// TwinCAT 3 PLC project CraneSimulation
// ProgramVersion: 3.1.4023.0
// libraries:
//   Tc2_Standard, * (Beckhoff Automation GmbH)
//   Tc2_System, * (Beckhoff Automation GmbH)
//   Tc3_Module, * (Beckhoff Automation GmbH)
//   VisuDialogs, * (System)
//   VisuSymbols,3.5.10.0,System
// project tree:
//   DUTs/ E_CraneMode.TcDUT, E_CraneStatus.TcDUT, E_ErrorModes.TcDUT, ST_CraneKinematics.TcDUT (not stored), ST_CraneParameters.TcDUT, ST_PistonOutOfBounds.TcDUT, ST_PistonRange.TcDUT, ST_StateVariables.TcDUT
//   / GlobalTextList.TcGTLO, PlcTask.TcTTO (not stored), Visualization Manager.TcVMO (not stored)
//   GVLs/ HMI.TcGVL, Inputs.TcGVL, Outputs.TcGVL, Parameters.TcGVL
//   POUs/ CraneSimulation.TcPOU, MAIN.TcPOU
//   POUs/Function blocks/ FB_AutomaticControl.TcPOU, FB_CheckPistonPosition.TcPOU, FB_CraneMode.TcPOU, FB_CraneStatus.TcPOU, FB_ManualControl.TcPOU, FB_MotionReferenceGenerator.TcPOU, FB_OpenLoopControl.TcPOU
//   POUs/Functions/ F_BarToPascal.TcPOU, F_BoomAngle.TcPOU, F_CheckPistonPosition.TcPOU, F_LminToSI.TcPOU, F_PistonDisplacementToBoomAngle.TcPOU, F_RadToDeg.TcPOU
//   VISUs/ CraneSimulationHMI.TcVIS

// ---- DUTs/E_CraneMode.TcDUT
{attribute 'qualified_only'}
{attribute 'strict'}
TYPE E_CraneMode :
(
	Manual,
	Automatic,
	NaN
);
END_TYPE

// ---- DUTs/E_CraneStatus.TcDUT
{attribute 'qualified_only'}
{attribute 'strict'}
TYPE E_CraneStatus :
(
	Error,
	Ready,
	Running,
	Stopping,
	PowerOff,
	Checking
);
END_TYPE

// ---- DUTs/E_ErrorModes.TcDUT
{attribute 'qualified_only'}
{attribute 'strict'}
TYPE E_ErrorModes :
(
	NaN,
	MaxLimit,
	MinLimit
);
END_TYPE

// ---- DUTs/ST_CraneParameters.TcDUT
TYPE ST_CraneParameters :
STRUCT
	fCyclicTime : LREAL := 0.01; //[s]
	fMaxVelocityLimit : LREAL := 0.05; //[m/s]
	fBoreArea : LREAL := 0.0033183;
	fAnnulusArea : LREAL := 0.0023562;
	fMaxFlowCapacity : LREAL := 30; //[l/min]
END_STRUCT
END_TYPE

// ---- DUTs/ST_PistonOutOfBounds.TcDUT
TYPE ST_PistonOutOfBounds :
STRUCT
	sNotActive : STRING := 'End Stop not active';
	sPistonMax : STRING := 'Piston has reached upper end stop';
	sPistonMin : STRING := 'Piston has reached lower end stop';
END_STRUCT
END_TYPE

// ---- DUTs/ST_PistonRange.TcDUT
TYPE ST_PistonRange :
STRUCT
	fPistonPosMax : REAL := 0.5;
	fPistonPosMin : REAL := 0.0;
END_STRUCT
END_TYPE

// ---- DUTs/ST_StateVariables.TcDUT
TYPE ST_StateVariables :
STRUCT
	bPower : BOOL;
	bStart : BOOL;
	bStop : BOOL;
	bRunning : BOOL := FALSE;
	bError : BOOL;
	bMode : BOOL;
	fTime : LREAL := 0.0;
END_STRUCT
END_TYPE

// ---- GVLs/HMI.TcGVL
{attribute 'qualified_only'}
VAR_GLOBAL
	fManualCylinderPositionReference : LREAL;
	sPistonEndStopMessage : STRING;
	fCylinderPositonReference : LREAL := 0.0;
	fCylinderVelocityReference : LREAL := 0.0;
	fBoomAngle : LREAL;
END_VAR

// ---- GVLs/Inputs.TcGVL
{attribute 'qualified_only'}
VAR_GLOBAL
	bOnSelector : BOOL;
	bAutoSelector : BOOL;
	bStartButton : BOOL;
	bStopButton : BOOL;
	fJoystickX : LREAL;
	fJoystickY : LREAL;
END_VAR

// ---- GVLs/Outputs.TcGVL
{attribute 'qualified_only'}
VAR_GLOBAL
	bStartLight : BOOL;
	bStopLight : BOOL;
	eCraneMode : E_CraneMode;
	eCraneStatus : E_CraneStatus;
	fOutputVelocity : LREAL;
END_VAR

// ---- GVLs/Parameters.TcGVL
{attribute 'qualified_only'}
VAR_GLOBAL
	fCyclicTime : REAL := 0.01;
	bSimulationRunning : BOOL := FALSE;
	stPistonRange : ST_PistonRange;
	stPistonOutOfBounds : ST_PistonOutOfBounds;
	stCraneKinematics : ST_CraneKinematics;
	stStateVariables : ST_StateVariables;
	stCraneParameters : ST_CraneParameters;
	eErrorModes : E_ErrorModes;
END_VAR

// ---- POUs/CraneSimulation.TcPOU
PROGRAM CraneSimulation
VAR
	fCyclicTime : LREAL := 0.01;
	
	fbCraneStatus : FB_CraneStatus;
	fbCraneMode : FB_CraneMode;
END_VAR

// Crane status state machine
fbCraneStatus(	bPower := Inputs.bOnSelector,
		 		bStart := Inputs.bStartButton, 
				bStop := Inputs.bStopButton, 
				bRunning := Parameters.stStateVariables.bRunning, 
				bError := Parameters.stStateVariables.bError,
				eCraneStatus => Outputs.eCraneStatus);

// Crane mode state machine
IF Parameters.stStateVariables.bRunning THEN
	fbCraneMode( 	bRunning := Parameters.stStateVariables.bRunning,
					bMode := Inputs.bAutoSelector,
					eCraneMode => Outputs.eCraneMode);
END_IF
	
// Calculate boom angle for visualization of simulation		
HMI.fBoomAngle := F_BoomAngle(	fCylinderX := HMI.fCylinderPositonReference);

// Simulation timer			
IF Parameters.stStateVariables.bRunning THEN
	Parameters.stStateVariables.fTime := Parameters.stStateVariables.fTime + fCyclicTime;
ELSE
	Parameters.stStateVariables.fTime := 0.0;
END_IF

END_PROGRAM

// ---- POUs/Function blocks/FB_CraneStatus.TcPOU
FUNCTION_BLOCK FB_CraneStatus
VAR_INPUT
	bPower : BOOL;
	bStart : BOOL;
	bStop : BOOL;
	bRunning : BOOL;
	bError : BOOL;
END_VAR
VAR_OUTPUT
	eCraneStatus : E_CraneStatus := E_CraneStatus.PowerOff;
END_VAR
VAR
END_VAR

//Status state machine
CASE eCraneStatus OF
	E_CraneStatus.PowerOff:
		IF bPower THEN
			eCraneStatus := E_CraneStatus.Checking;
		END_IF	
	
	E_CraneStatus.Error:
		Outputs.bStopLight := TRUE;
		
		IF NOT bError THEN
			eCraneStatus := E_CraneStatus.Checking;
		END_IF
		
	E_CraneStatus.Checking:
		Outputs.bStopLight := FALSE;
		Outputs.bStartLight := FALSE;
		
		IF (NOT bError) THEN
			eCraneStatus := E_CraneStatus.Ready;
		ELSE
			eCraneStatus := E_CraneStatus.Error;
		END_IF
		
		IF bPower AND NOT bError THEN
			eCraneStatus := E_CraneStatus.Ready;
		ELSE
			eCraneStatus := E_CraneStatus.PowerOff;
		END_IF
		
	E_CraneStatus.Ready:
		IF bStart AND bPower AND NOT(bError) THEN
			Parameters.stStateVariables.bRunning := TRUE;
			Parameters.stStateVariables.bStart := FALSE;
			eCraneStatus := E_CraneStatus.Running;
		END_IF	
		
		IF  NOT(bPower) OR bError THEN
			eCraneStatus := E_CraneStatus.Checking;
		END_IF	
		
	E_CraneStatus.Running:
		Outputs.bStartLight := TRUE;
		
		F_CheckPistonPosition();
		
		IF bStop THEN
			eCraneStatus := E_CraneStatus.Stopping;
		END_IF
		
		IF bError OR NOT bRunning OR NOT bPOWER THEN
			eCraneStatus := E_CraneStatus.Checking;
		END_IF
		
	E_CraneStatus.Stopping:
		Parameters.stStateVariables.bRunning := FALSE;
		Parameters.stStateVariables.bStart := FALSE;
		Outputs.bStopLight := TRUE;
	
		IF NOT bRunning OR bPower OR bError THEN
			eCraneStatus := E_CraneStatus.Checking;
		END_IF
	ELSE
		eCraneStatus := E_CraneStatus.Checking;
		
END_CASE

END_FUNCTION_BLOCK

// ---- POUs/Functions/F_CheckPistonPosition.TcPOU
FUNCTION F_CheckPistonPosition : E_ErrorModes
VAR_INPUT
END_VAR
VAR
END_VAR

// Check if piston is out of bounds
IF HMI.fCylinderPositonReference > Parameters.stPistonRange.fPistonPosMax THEN
	HMI.fCylinderPositonReference := Parameters.stPistonRange.fPistonPosMax;	
	HMI.sPistonEndStopMessage := Parameters.stPistonOutOfBounds.sPistonMax;
	Parameters.eErrorModes := E_ErrorModes.MaxLimit;
	HMI.sPistonEndStopMessage := Parameters.stPistonOutOfBounds.sPistonMax;
	Parameters.stStateVariables.fTime := 0.0;
ELSIF HMI.fCylinderPositonReference < Parameters.stPistonRange.fPistonPosMin  THEN
	HMI.fCylinderPositonReference := Parameters.stPistonRange.fPistonPosMin;
	Parameters.eErrorModes := E_ErrorModes.MinLimit;
	HMI.sPistonEndStopMessage := Parameters.stPistonOutOfBounds.sPistonMin;
	Parameters.stStateVariables.fTime := 0.0;
ELSE
	HMI.sPistonEndStopMessage := Parameters.stPistonOutOfBounds.sNotActive;
	Parameters.eErrorModes := E_ErrorModes.NaN;
END_IF

END_FUNCTION

// ---- POUs/Function blocks/FB_CraneMode.TcPOU
FUNCTION_BLOCK FB_CraneMode
VAR_INPUT
	bRunning : BOOL := FALSE; 
	bMode : BOOL := FALSE; //False for manual, true for automatic.
END_VAR
VAR_OUTPUT
	eCraneMode : E_CraneMode := E_CraneMode.Manual;
END_VAR
VAR
	fbManualControl : FB_ManualControl;
	fbAutomaticControl : FB_AutomaticControl;
END_VAR

CASE eCraneMode OF
	E_CraneMode.Manual:
		IF bMode THEN
			Parameters.stStateVariables.fTime := 0.0;
			eCraneMode := E_CraneMode.Automatic;
		ELSE
			fbManualControl();
		END_IF
		
	E_CraneMode.Automatic:
		IF NOT bMode THEN
			Parameters.stStateVariables.fTime := 0.0;
			eCraneMode := E_CraneMode.Manual;
		ELSE
			fbAutomaticControl();
		END_IF
		
	E_CraneMode.NaN:
		IF NOT bMode AND bRunning THEN
			eCraneMode := E_CraneMode.Manual;
		ELSIF bMode AND bRunning THEN
			eCraneMode := E_CraneMode.Automatic;
		END_IF
END_CASE

END_FUNCTION_BLOCK

// ---- POUs/Function blocks/FB_ManualControl.TcPOU
FUNCTION_BLOCK FB_ManualControl
VAR_INPUT
END_VAR
VAR_OUTPUT
	fVelocityFeedForwardControlOutput : LREAL;
END_VAR
VAR
	fNormalizedJoystickY : LREAL;
	fbOpenLoopControl : FB_OpenLoopControl; 
	bEnable : BOOL := TRUE;
END_VAR

CASE Parameters.eErrorModes OF
	E_ErrorModes.MaxLimit:
		IF Inputs.fJoystickY > 0.0 THEN
			Inputs.fJoystickY := 0.0;
		END_IF
	E_ErrorModes.MinLimit:
		IF Inputs.fJoystickY < 0.0 THEN
			Inputs.fJoystickY := 0.0;
		END_IF
END_CASE 

fNormalizedJoystickY := Inputs.fJoystickY*Parameters.stCraneParameters.fMaxVelocityLimit;

fbOpenLoopControl(
	bEnable := bEnable,
	stParam := Parameters.stCraneParameters,
	fInput_ms := fNormalizedJoystickY,
	fMaxValveFlow_lmin := Parameters.stCraneParameters.fMaxFlowCapacity,
	fNormalizedOutput => Outputs.fOutputVelocity
);

HMI.fCylinderPositonReference := Outputs.fOutputVelocity * 1/2*(Parameters.stStateVariables.fTime*Parameters.stStateVariables.fTime);

END_FUNCTION_BLOCK

// ---- POUs/Function blocks/FB_OpenLoopControl.TcPOU
FUNCTION_BLOCK FB_OpenLoopControl
VAR_INPUT
	bEnable : BOOL;
	fInput_ms : LREAL;
	fMaxValveFlow_lmin : LREAL;
	stParam : ST_CraneParameters;
END_VAR
VAR_OUTPUT
	fNormalizedOutput: LREAL;
END_VAR
VAR
	fFlowReference_m3s : LREAL;
	fM3sToLmin : LREAL := 60000;
END_VAR

IF fInput_ms >= 0.0 THEN 
    fFlowReference_m3s := stparam.fBoreArea * fInput_ms;
ELSE 
    fFlowReference_m3s := fInput_ms * stParam.fAnnulusArea;
END_IF;

IF bEnable THEN 
    fNormalizedOutput := (fM3sToLmin * fFlowReference_m3s) / fMaxValveFlow_lmin;
ELSE 
    fNormalizedOutput := 0.0;
END_IF;

END_FUNCTION_BLOCK

// ---- POUs/Function blocks/FB_AutomaticControl.TcPOU
FUNCTION_BLOCK FB_AutomaticControl
VAR_INPUT
END_VAR
VAR_OUTPUT
END_VAR
VAR
	fbMotionReferenceGenerator : FB_MotionReferenceGenerator;
END_VAR

fbMotionReferenceGenerator(
	bEnable := TRUE,
	fStartPosition_m := 0.0,
	fStartVelocity_m := 0.0,
	fPositionSetpoint_m := 0.4,
	fVelocitySetpoint_m := 0.05,
	fTimeBeforeStarting_s := 2,
	fRampTime_s := 1,
	fHoldPositionTime_s := 3,
	fClock_s := Parameters.stStateVariables.fTime, 
	fVelocityReference_m => Outputs.fOutputVelocity,
	fPositionReference_m => HMI.fCylinderPositonReference
);

END_FUNCTION_BLOCK

// ---- POUs/Function blocks/FB_MotionReferenceGenerator.TcPOU
FUNCTION_BLOCK FB_MotionReferenceGenerator
VAR_INPUT
	bEnable: BOOL;
	fStartPosition_m: LREAL;
	fStartVelocity_m: LREAL;
	fPositionSetpoint_m: LREAL;
	fVelocitySetpoint_m: LREAL;
	fTimeBeforeStarting_s: LREAL;
	fRampTime_s: LREAL;
	fHoldPositionTime_s: LREAL;
	fClock_s: LREAL;
END_VAR
VAR_OUTPUT
	fPositionReference_m: LREAL;
	fVelocityReference_m: LREAL;
	fTotalMotionTime_s: LREAL;
	fErrorSignal: LREAL;
END_VAR
VAR
	Error: DINT;
	slopeExt: LREAL;
	tHold: LREAL;
	x1: LREAL;
	x4: LREAL;
	rtb_Saturation3: LREAL;
	x1_tmp: LREAL;
	x1_tmp_tmp: LREAL;
	x4_tmp: LREAL;
	x4_tmp_tmp: LREAL;
	x4_tmp_tmp_0: LREAL;
	x4_tmp_tmp_1: LREAL;
	x1_tmp_0: LREAL;
END_VAR


(* Outputs for Atomic SubSystem: '<Root>/FB_MotionReferenceGenerator' *)
(* Saturate: '<S1>/Saturation2' *)

IF fVelocitySetpoint_m > 0.05 THEN 
    fPositionReference_m := 0.05;
ELSIF fVelocitySetpoint_m >= 0.0 THEN 
    fPositionReference_m := fVelocitySetpoint_m;
ELSE 
    fPositionReference_m := 0.0;
END_IF;

(* End of Saturate: '<S1>/Saturation2' *)


(* Saturate: '<S1>/Saturation3' *)

IF fPositionSetpoint_m > 0.45 THEN 
    rtb_Saturation3 := 0.45;
ELSIF fPositionSetpoint_m >= 0.0 THEN 
    rtb_Saturation3 := fPositionSetpoint_m;
ELSE 
    rtb_Saturation3 := 0.0;
END_IF;

(* End of Saturate: '<S1>/Saturation3' *)


(* MATLAB Function: '<S1>/WaveSignal' *)
(* MATLAB Function 'FB_MotionReferenceGenerator/WaveSignal': '<S2>:1' *)
(* '<S2>:1:2' x_SP = x_ref - x0; *)
(* '<S2>:1:3' vs=v_ref; *)
(* '<S2>:1:4' slopeExt=v0-vs; *)
slopeExt := fStartVelocity_m - fPositionReference_m;
(* '<S2>:1:5' slopeRetr=-vs-v0; *)
(* '<S2>:1:7' as = vs/tRamp; *)
(* '<S2>:1:8' s_acc=(vs^2-v0^2)/as; *)
(* '<S2>:1:10' tHold=(x_SP-s_acc)/vs; *)
tHold := ((rtb_Saturation3 - fStartPosition_m) - (((fPositionReference_m * fPositionReference_m) - (fStartVelocity_m * fStartVelocity_m)) / (fPositionReference_m / fRampTime_s))) / fPositionReference_m;
(* '<S2>:1:12' if tHold < 0 *)

IF tHold < 0.0 THEN 
    (* '<S2>:1:13' Error = 1; *)
    Error := 1;
ELSE 
    (* '<S2>:1:14' else *)
    (* '<S2>:1:15' Error = 0; *)
    Error := 0;
END_IF;

(* '<S2>:1:18' t1=tRamp; *)
(* '<S2>:1:19' t2=tHold; *)
(* '<S2>:1:20' t3=tRamp; *)
(* '<S2>:1:21' t4=tWait; *)
(* '<S2>:1:22' t5=t1; *)
(* '<S2>:1:23' t6=t2; *)
(* '<S2>:1:24' t7=t3; *)
(* '<S2>:1:26' x = x0; *)
(* '<S2>:1:27' x1 = x0 + v0*((t0+t1)-t0)-(slopeExt/t1)*((t0+t1)-t0)^2/2; *)
x1_tmp_tmp := fTimeBeforeStarting_s + fRampTime_s;
x1_tmp := x1_tmp_tmp - fTimeBeforeStarting_s;
x1_tmp_0 := slopeExt / fRampTime_s;
x1 := ((x1_tmp * fStartVelocity_m) + fStartPosition_m) - ((x1_tmp_0 * (x1_tmp * x1_tmp)) / 2.0);
(* '<S2>:1:28' x2 = x1 + vs*((t0+t1+t2)-(t0+t1)); *)
(* '<S2>:1:29' x4 = x_ref - v0*((t0+t1+t2+t3+t4+t5)-(t0+t1+t2+t3+t4))+(slopeRetr/t5)*((t0+t1+t2+t3+t4+t5)-(t0+t1+t2+t3+t4))^2/2; *)
x4_tmp_tmp := x1_tmp_tmp + tHold;
x4_tmp_tmp_0 := x4_tmp_tmp + fRampTime_s;
x4_tmp := x4_tmp_tmp_0 + fHoldPositionTime_s;
x4_tmp_tmp_1 := x4_tmp + fRampTime_s;
x4 := x4_tmp_tmp_1 - x4_tmp;
x1_tmp := (( -fPositionReference_m) - fStartVelocity_m) / fRampTime_s;
x4 := (rtb_Saturation3 - (x4 * fStartVelocity_m)) + ((x1_tmp * (x4 * x4)) / 2.0);
(* '<S2>:1:30' x5 = x4-vs*((t0+t1+t2+t3+t4+t5+t6)-(t0+t1+t2+t3+t4+t5)); *)
(* '<S2>:1:32' if Error == 1 *)

IF Error = 1 THEN 
    (* '<S2>:1:33' x = x0; *)
    rtb_Saturation3 := fStartPosition_m;
    (* '<S2>:1:34' v = v0; *)
    fPositionReference_m := fStartVelocity_m;
ELSIF (fClock_s >= 0.0) AND (fClock_s < fTimeBeforeStarting_s) THEN 
    (* '<S2>:1:35' elseif t>=0 && t<t0 *)
    (* '<S2>:1:36' x = x0; *)
    rtb_Saturation3 := fStartPosition_m;
    (* '<S2>:1:37' v = v0; *)
    fPositionReference_m := fStartVelocity_m;
ELSIF (fClock_s >= fTimeBeforeStarting_s) AND (fClock_s < x1_tmp_tmp) THEN 
    (* '<S2>:1:38' elseif t>=t0 && t<(t0+t1) *)
    (* '<S2>:1:39' x = x0 + v0*(t-t0)-(slopeExt/t1)*(t-t0)^2/2; *)
    x4_tmp_tmp_0 := fClock_s - fTimeBeforeStarting_s;
    rtb_Saturation3 := ((x4_tmp_tmp_0 * fStartVelocity_m) + fStartPosition_m) - ((x1_tmp_0 * (x4_tmp_tmp_0 * x4_tmp_tmp_0)) / 2.0);
    (* '<S2>:1:40' v = v0-(slopeExt/t1)*(t-t0); *)
    fPositionReference_m := fStartVelocity_m - (x1_tmp_0 * x4_tmp_tmp_0);
ELSIF (fClock_s >= x1_tmp_tmp) AND (fClock_s < x4_tmp_tmp) THEN 
    (* '<S2>:1:41' elseif t>=(t0+t1) && t<(t0+t1+t2) *)
    (* '<S2>:1:42' x = x1 + vs*(t-(t0+t1)); *)
    rtb_Saturation3 := ((fClock_s - x1_tmp_tmp) * fPositionReference_m) + x1;
    (* '<S2>:1:43' v = vs; *)
ELSIF (fClock_s >= x4_tmp_tmp) AND (fClock_s < x4_tmp_tmp_0) THEN 
    (* '<S2>:1:44' elseif t>=(t0+t1+t2) && t<(t0+t1+t2+t3) *)
    (* '<S2>:1:45' x = x2+vs*(t-(t0+t1+t2))+(slopeExt/t3)*(t-(t0+t1+t2))^2/2; *)
    x4_tmp_tmp_0 := fClock_s - x4_tmp_tmp;
    rtb_Saturation3 := ((((x4_tmp_tmp - x1_tmp_tmp) * fPositionReference_m) + x1) + (x4_tmp_tmp_0 * fPositionReference_m)) + ((x1_tmp_0 * (x4_tmp_tmp_0 * x4_tmp_tmp_0)) / 2.0);
    (* '<S2>:1:46' v = vs+(slopeExt/t3)*(t-(t0+t1+t2)); *)
    fPositionReference_m := (x4_tmp_tmp_0 * (slopeExt / fRampTime_s)) + fPositionReference_m;
ELSIF (fClock_s >= x4_tmp_tmp_0) AND (fClock_s < x4_tmp) THEN 
    (* '<S2>:1:47' elseif t>=(t0+t1+t2+t3) && t<(t0+t1+t2+t3+t4) *)
    (* '<S2>:1:48' x = x_ref; *)
    (* '<S2>:1:49' v = v0; *)
    fPositionReference_m := fStartVelocity_m;
ELSIF (fClock_s >= x4_tmp) AND (fClock_s < x4_tmp_tmp_1) THEN 
    (* '<S2>:1:50' elseif t>=(t0+t1+t2+t3+t4) && t<(t0+t1+t2+t3+t4+t5) *)
    (* '<S2>:1:51' x = x_ref - v0*(t-(t0+t1+t2+t3+t4))+(slopeRetr/t5)*(t-(t0+t1+t2+t3+t4))^2/2; *)
    slopeExt := fClock_s - x4_tmp;
    rtb_Saturation3 := (rtb_Saturation3 - (slopeExt * fStartVelocity_m)) + ((x1_tmp * (slopeExt * slopeExt)) / 2.0);
    (* '<S2>:1:52' v = v0+(slopeRetr/t5)*(t-(t0+t1+t2+t3+t4)); *)
    fPositionReference_m := (slopeExt * x1_tmp) + fStartVelocity_m;
ELSE 
    rtb_Saturation3 := x4_tmp_tmp_1 + tHold;

    IF (fClock_s >= x4_tmp_tmp_1) AND (fClock_s < rtb_Saturation3) THEN 
        (* '<S2>:1:53' elseif t>=(t0+t1+t2+t3+t4+t5) && t<(t0+t1+t2+t3+t4+t5+t6) *)
        (* '<S2>:1:54' x = x4-vs*(t-(t0+t1+t2+t3+t4+t5)); *)
        rtb_Saturation3 := x4 - ((fClock_s - x4_tmp_tmp_1) * fPositionReference_m);
        (* '<S2>:1:55' v = -vs; *)
        fPositionReference_m :=  -fPositionReference_m;
    ELSIF (fClock_s >= rtb_Saturation3) AND (fClock_s < (rtb_Saturation3 + fRampTime_s)) THEN 
        (* '<S2>:1:56' elseif t>=(t0+t1+t2+t3+t4+t5+t6) && t<(t0+t1+t2+t3+t4+t5+t6+t7) *)
        (* '<S2>:1:57' x = x5-vs*(t-(t0+t1+t2+t3+t4+t5+t6))-(slopeRetr/t3)*(t-(t0+t1+t2+t3+t4+t5+t6))^2/2; *)
        x4_tmp_tmp_0 := fClock_s - rtb_Saturation3;
        rtb_Saturation3 := ((x4 - ((rtb_Saturation3 - x4_tmp_tmp_1) * fPositionReference_m)) - (x4_tmp_tmp_0 * fPositionReference_m)) - ((x1_tmp * (x4_tmp_tmp_0 * x4_tmp_tmp_0)) / 2.0);
        (* '<S2>:1:58' v = -vs-(slopeRetr/t3)*(t-(t0+t1+t2+t3+t4+t5+t6)); *)
        fPositionReference_m := ( -fPositionReference_m) - (x4_tmp_tmp_0 * x1_tmp);
    ELSE 
        (* '<S2>:1:59' else *)
        (* '<S2>:1:60' x = x0; *)
        rtb_Saturation3 := fStartPosition_m;
        (* '<S2>:1:61' v = v0; *)
        fPositionReference_m := fStartVelocity_m;
    END_IF;

END_IF;

(* Switch: '<S1>/Switch' *)
(* '<S2>:1:64' T = t0+t1+t2+t3+t4+t5+t6+t7; *)

IF  NOT bEnable THEN 
    fPositionReference_m := fStartVelocity_m;
END_IF;

(* End of Switch: '<S1>/Switch' *)


(* Saturate: '<S1>/Saturation' *)

IF fPositionReference_m > 0.05 THEN 
    (* Outport: '<Root>/fVelocityReference_m' *)
    fVelocityReference_m := 0.05;
ELSIF fPositionReference_m >= -0.05 THEN 
    (* Outport: '<Root>/fVelocityReference_m' *)
    fVelocityReference_m := fPositionReference_m;
ELSE 
    (* Outport: '<Root>/fVelocityReference_m' *)
    fVelocityReference_m := -0.05;
END_IF;

(* End of Saturate: '<S1>/Saturation' *)


(* Switch: '<S1>/Switch1' *)

IF bEnable THEN 
    fPositionReference_m := rtb_Saturation3;
ELSE 
    fPositionReference_m := fStartPosition_m;
END_IF;

(* End of Switch: '<S1>/Switch1' *)


(* Saturate: '<S1>/Saturation1' *)

IF fPositionReference_m > 0.45 THEN 
    (* Outport: '<Root>/fPositionReference_m' *)
    fPositionReference_m := 0.45;
ELSIF fPositionReference_m < 0.0 THEN 
    (* Outport: '<Root>/fPositionReference_m' *)
    fPositionReference_m := 0.0;
END_IF;

(* End of Saturate: '<S1>/Saturation1' *)


(* Outport: '<Root>/fTotalMotionTime_s' incorporates:
 *  MATLAB Function: '<S1>/WaveSignal' *)
fTotalMotionTime_s := ((((((fTimeBeforeStarting_s + fRampTime_s) + tHold) + fRampTime_s) + fHoldPositionTime_s) + fRampTime_s) + tHold) + fRampTime_s;
(* Outport: '<Root>/fErrorSignal' incorporates:
 *  MATLAB Function: '<S1>/WaveSignal' *)
fErrorSignal := DINT_TO_LREAL(Error);
(* End of Outputs for SubSystem: '<Root>/FB_MotionReferenceGenerator' *)

END_FUNCTION_BLOCK

// ---- POUs/Functions/F_BoomAngle.TcPOU
FUNCTION F_BoomAngle : LREAL
VAR_INPUT
	fCylinderX : LREAL;
END_VAR
VAR_OUTPUT
END_VAR
VAR
	fAngleRad : LREAL;
END_VAR

fAngleRad := F_PistonDisplacementToBoomAngle(xCyl := fCylinderX);
F_BoomAngle := F_RadToDeg(fRad := fAngleRad);

END_FUNCTION

// ---- POUs/Functions/F_PistonDisplacementToBoomAngle.TcPOU
FUNCTION F_PistonDisplacementToBoomAngle : LREAL
VAR_INPUT
	xCyl : LREAL;
END_VAR
VAR
	AB : LREAL;
	AC : LREAL;
	BC : LREAL;
	alpha1 : LREAL;
	alpha2 : LREAL;
	theta1 : LREAL;
	AB2 : LREAL;
	AC2 : LREAL;
	BC2 : LREAL;
END_VAR

AB := SQRT(ABS(Parameters.stCraneKinematics.ABx)*ABS(Parameters.stCraneKinematics.ABx) + ABS(Parameters.stCraneKinematics.ABy)*ABS(Parameters.stCraneKinematics.ABy));
AC := SQRT(ABS(Parameters.stCraneKinematics.ACx)*ABS(Parameters.stCraneKinematics.ACx) + ABS(Parameters.stCraneKinematics.ACy)*ABS(Parameters.stCraneKinematics.ACy));

BC := 0.77222 + xCyl;

alpha1 := ATAN(ABS(Parameters.stCraneKinematics.ACy)/ ABS(Parameters.stCraneKinematics.ACx));
alpha2 := ATAN(ABS(Parameters.stCraneKinematics.ABy)/ ABS(Parameters.stCraneKinematics.ABx));

AB2 := ABS(AB)*ABS(AB);
AC2 := ABS(AC)*ABS(AC);
BC2 := ABS(BC)*ABS(BC);

theta1 := ACOS( (AB2 + AC2 - BC2) / (2 * ABS(AB) * ABS(AC)) ) - alpha2 + alpha1;

F_PistonDisplacementToBoomAngle := theta1;

END_FUNCTION

// ---- POUs/Functions/F_RadToDeg.TcPOU
FUNCTION F_RadToDeg : LREAL
VAR_INPUT
	fRad :LREAL;
END_VAR
VAR
END_VAR

F_RadToDeg := fRad * (180/PI);

END_FUNCTION

// ---- POUs/Function blocks/FB_CheckPistonPosition.TcPOU
FUNCTION_BLOCK FB_CheckPistonPosition
VAR_INPUT
END_VAR
VAR_OUTPUT
END_VAR
VAR
END_VAR

// Check if piston is out of bounds
IF HMI.fCylinderPositonReference > Parameters.stPistonRange.fPistonPosMax THEN
	HMI.fCylinderPositonReference := Parameters.stPistonRange.fPistonPosMax;	
	HMI.sPistonEndStopMessage := Parameters.stPistonOutOfBounds.sPistonMax;
	Parameters.eErrorModes := E_ErrorModes.MaxLimit;
	HMI.sPistonEndStopMessage := Parameters.stPistonOutOfBounds.sPistonMax;
ELSIF HMI.fCylinderPositonReference < Parameters.stPistonRange.fPistonPosMin  THEN
	HMI.fCylinderPositonReference := Parameters.stPistonRange.fPistonPosMin;
	Parameters.eErrorModes := E_ErrorModes.MinLimit;
	HMI.sPistonEndStopMessage := Parameters.stPistonOutOfBounds.sPistonMin;
ELSE
	HMI.sPistonEndStopMessage := Parameters.stPistonOutOfBounds.sNotActive;
	Parameters.eErrorModes := E_ErrorModes.NaN;
END_IF

END_FUNCTION_BLOCK

// ---- POUs/Functions/F_BarToPascal.TcPOU
FUNCTION F_BarToPascal : LREAL
VAR_INPUT
	fBar : LREAL;
END_VAR
VAR
END_VAR

F_BarToPascal := fBar*1E5;

END_FUNCTION

// ---- POUs/Functions/F_LminToSI.TcPOU
FUNCTION F_LminToSI : LREAL
VAR_INPUT
	fLmin : LREAL;
END_VAR
VAR
END_VAR

F_LminToSI := fLmin / 60000;

END_FUNCTION

// ---- POUs/MAIN.TcPOU
PROGRAM MAIN
VAR
END_VAR

CraneSimulation();

END_PROGRAM

// ---- GlobalTextList.TcGTLO
TEXTLIST GlobalTextList
  99 = '%..1f'
  219 = '%.01f'
  275 = '%.1f'
  130 = '%.2f'
  940 = '%0.01f'
  283 = '%0.1f'
  831 = '%1.f'
  223 = '%f'
  819 = '%s'
  133 = '1'
  655 = 'AUTO'
  90 = 'Crane error message: %s'
  502 = 'Crane message:'
  113 = 'Crane message: %s'
  457 = 'Crane mode: %s'
  517 = 'Crane status: %s'
  957 = 'Crane staus: %s'
  127 = 'Cylinder position'
  166 = 'Cylinder position reference:'
  995 = 'Cylinder Position Reference: %f [m]'
  983 = 'Cylinder position:'
  582 = 'Cylinder velocity reference:'
  25 = 'Cylinder Velocity Reference: %f [m/s]'
  222 = 'Cylinder velocity:'
  0 = 'dsafasd'
  280 = 'ENABLE'
  496 = 'ENABLE\t\tStart \t\tAuto '
  444 = 'ENABLE\t\tStart \tAuto '
  752 = 'ENABLE\t\tStart Simulation\t\t\t Auto '
  850 = 'ERROR'
  204 = 'FAULT'
  961 = 'JOYSTICK Y'
  829 = 'Joystick Y:'
  689 = 'MANUAL'
  362 = 'Manual cylinder position reference:'
  782 = 'Manual sylinder position reference:'
  648 = 'Manual ylinder position reference:'
  188 = 'Mode'
  65 = 'OFF'
  629 = 'ON'
  911 = 'POWER'
  581 = 'REAL'
  526 = 'RUNNING'
  503 = 'Simulation'
  38 = 'Simulation time: '
  680 = 'Simulation time: %f'
  741 = 'Simulation time: %f s'
  136 = 'Simulation time: %i'
  413 = 'START'
  795 = 'Status'
  696 = 'STOP'
END_TEXTLIST

// ---- VISUs/CraneSimulationHMI.TcVIS
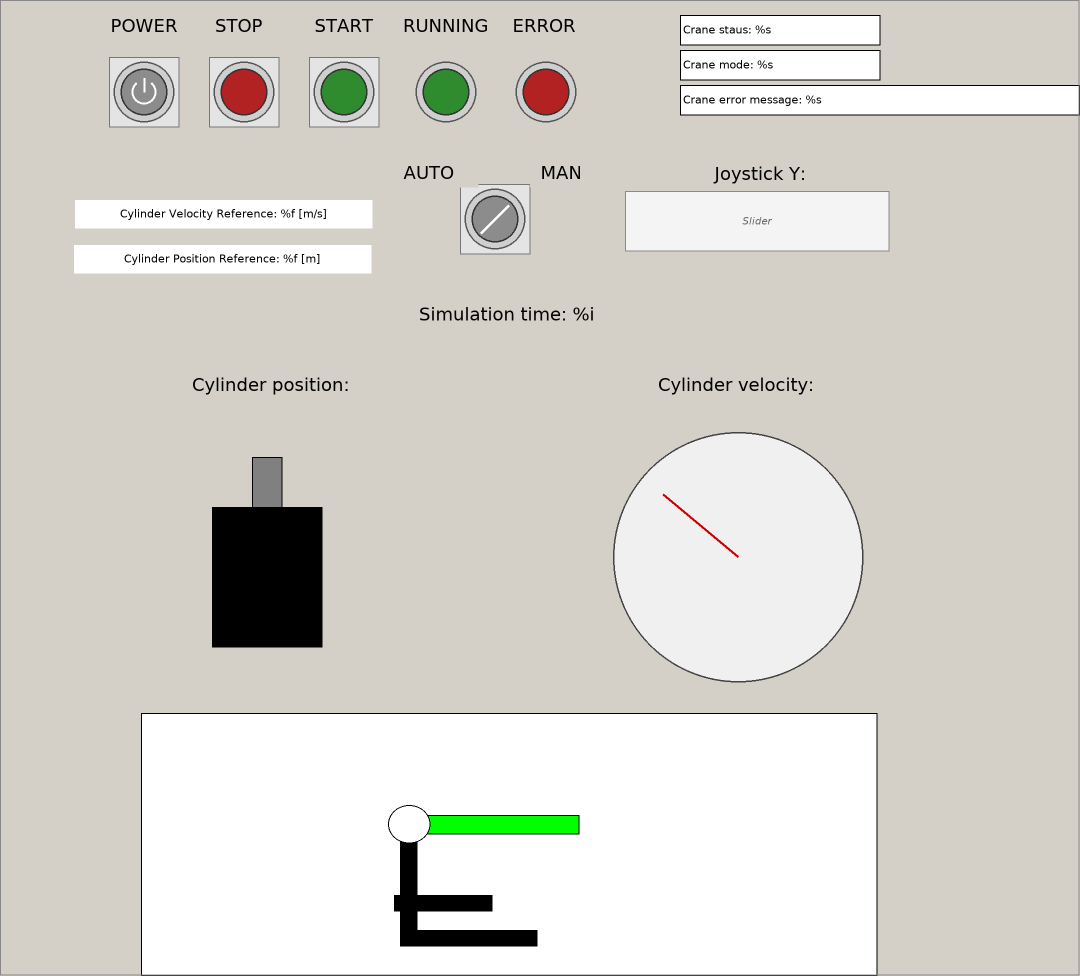
VISUALIZATION CraneSimulationHMI  // 1080x976
    PowerSwitch (109,57 70x70), variable: Inputs.bOnSelector, behaviour: TOGGLE, style: Switch-PowerSwitch-Gray
    RotarySwitch (460,184 70x70), variable: Inputs.bAutoSelector, behaviour: TOGGLE, style: Switch-RotarySwitch-Gray
    PushSwitch (309,57 70x70), variable: Inputs.bStartButton, behaviour: TOGGLE, style: Switch-PushSwitch-Green
    Rectangle (94,12 100x28), "POWER"
    Rectangle (294,12 100x28), "START"
    Rectangle (380,159 98x28), "AUTO"
    Rectangle (530,159 98x28), "MANUAL"
    Lamp1 (411,57 70x70), variable: Outputs.bStartLight, style: Lamp-Lamp1-Green
    Rectangle (396,12 100x28), "RUNNING"
    Rectangle (239,301 536x27), "Simulation time: %i", text variable: Parameters.stStateVariables.fTime
    Meter360 (613,432 250x250), value: Outputs.fOutputVelocity, style: Meter-Meter360-Gray, scale format: %.2f, scale -0.05..0.05
    Rectangle (182,372 178x26), "Cylinder position:"
    Rectangle (647,372 178x26), "Cylinder velocity:"
    Rectangle (680,85 400x30), "Crane error message: %s", text variable: HMI.sPistonEndStopMessage
    Rectangle (680,50 200x30), "Crane mode: %s", text variable: Outputs.eCraneMode
    Rectangle (680,15 200x30), "Crane staus: %s", text variable: Outputs.eCraneStatus
    Rectangle (252,457 30x180)
        p2738717112: -HMI.fCylinderPositonReference*100
    Rectangle (212,507 110x140)
    Textfield (73,244 299x30), "Cylinder Position Reference: %f [m]", text variable: HMI.fCylinderPositonReference
    Textfield (74,199 299x30), "Cylinder Velocity Reference: %f [m/s]", text variable: HMI.fCylinderVelocityReference
        OnMouseClick: write the text variable via Default
    PushSwitch (209,57 70x70), variable: Inputs.bStopButton, behaviour: TAP, style: Switch-PushSwitch-Red
    Rectangle (189,12 100x28), "STOP"
    Rectangle (141,713 736x263)
    Rectangle (400,930 137x16)
    Rectangle (400,810 17x130)
    Rectangle (409,815 170x19), angle 5
        p2858320360: -HMI.fBoomAngle
    Ellipse (388,805 42x38)
    Lamp1 (511,57 70x70), variable: Outputs.bStopLight, style: Lamp-Lamp1-Red
    Rectangle (494,12 100x28), "ERROR"
    Rectangle (394,895 98x16), angle 43
    Rectangle (580,162 361x24), "Joystick Y:"
    Slider (625,191 264x60), variable: Inputs.fJoystickY, scale -1..1
END_VISUALIZATION
